(* IEC 61131-3 sources: AXOpen/src/components.elements/ctrl/test, 10 files *)

(* ---- AxoAiTests.st ---- *)
USING AxUnit;
USING AXOpen.Components.Elements;
USING AXOpen.Core;
USING AXOpen.Rtc;
USING AXOpen.Logging;

NAMESPACE AXOpen.Components.Elements.Tests

    {TestFixture}
    {S7.extern=ReadWrite}
    CLASS AxoAiTests
        VAR
            context : TestContext;
            _testAxoAi : AxoAi;
            _signal : DINT;

            _done : BOOL;
        END_VAR

        {Test(signal := 100, required := 100)}
        {Test(signal := 50, required := 50)}
        {Test(signal := 0, required := 0)}
        {Test(signal := -50, required := -50)}
        {Test(signal := -100, required := -100)}
        METHOD PUBLIC RoundedRawRoundedReal
            VAR_INPUT
                signal : DINT;
                required : REAL;
            END_VAR

            context.Open();

            _testAxoAi._config.RawLow := -100;
            _testAxoAi._config.RawHigh := 100;
            _testAxoAi._config.RealLow := -100;
            _testAxoAi._config.RealHigh := 100;
            _testAxoAi._config.Gain := 1;
            _testAxoAi._config.Offset := 0;
            _signal := signal;

            _testAxoAi.Run(context.SignalParent, _signal);

            AxUnit.Assert.Equal(TRUE, TO_DINT(required) = TO_DINT(_testAxoAi._scaled));

            context.Close();

        END_METHOD

        {Test(signal := 32767, required := 100)}
        {Test(signal := 16384, required := 50)}
        {Test(signal := 0, required := 0)}
        METHOD PUBLIC UnsignedRawTest
            VAR_INPUT
                signal : DINT;
                required : REAL;
            END_VAR

            context.Open();

            _testAxoAi._config.RawLow := 0;
            _testAxoAi._config.RawHigh := 32767;
            _testAxoAi._config.RealLow := 0;
            _testAxoAi._config.RealHigh := 100;
            _testAxoAi._config.Gain := 1;
            _testAxoAi._config.Offset := 0;
            _signal := signal;

            _testAxoAi.Run(context.SignalParent, _signal);

            AxUnit.Assert.Equal(TRUE, TO_DINT(required) = TO_DINT(_testAxoAi._scaled));

            context.Close();

        END_METHOD

        {Test(signal := 32767, required := 100)}
        {Test(signal := 0, required := 50)}
        {Test(signal := -32768, required := 0)}
        METHOD PUBLIC SignedRawTest
            VAR_INPUT
                signal : DINT;
                required : REAL;
            END_VAR

            context.Open();

            _testAxoAi._config.RawLow := -32768;
            _testAxoAi._config.RawHigh := 32767;
            _testAxoAi._config.RealLow := 0;
            _testAxoAi._config.RealHigh := 100;
            _testAxoAi._config.Gain := 1;
            _testAxoAi._config.Offset := 0;
            _signal := signal;

            _testAxoAi.Run(context.SignalParent, _signal);

            AxUnit.Assert.Equal(TRUE, TO_DINT(required) = TO_DINT(_testAxoAi._scaled));

            context.Close();

        END_METHOD

        {Test(signal := 32767, required := 100)}
        {Test(signal := 16384, required := 75)}
        {Test(signal := 0, required := 50)}
        METHOD PUBLIC UnsignedRaw_RealOffsetTest
            VAR_INPUT
                signal : DINT;
                required : REAL;
            END_VAR

            context.Open();

            _testAxoAi._config.RawLow := 0;
            _testAxoAi._config.RawHigh := 32767;
            _testAxoAi._config.RealLow := 50;
            _testAxoAi._config.RealHigh := 100;
            _testAxoAi._config.Gain := 1;
            _testAxoAi._config.Offset := 0;
            _signal := signal;

            _testAxoAi.Run(context.SignalParent, _signal);

            AxUnit.Assert.Equal(TRUE, TO_DINT(required) = TO_DINT(_testAxoAi._scaled));

            context.Close();

        END_METHOD

        {Test(signal := 32767, required := 100)}
        {Test(signal := 0, required := 75)}
        {Test(signal := -32768, required := 50)}
        METHOD PUBLIC SignedRaw_RealOffsetTest
            VAR_INPUT
                signal : DINT;
                required : REAL;
            END_VAR

            context.Open();

            _testAxoAi._config.RawLow := -32768;
            _testAxoAi._config.RawHigh := 32767;
            _testAxoAi._config.RealLow := 50;
            _testAxoAi._config.RealHigh := 100;
            _testAxoAi._config.Gain := 1;
            _testAxoAi._config.Offset := 0;
            _signal := signal;

            _testAxoAi.Run(context.SignalParent, _signal);

            AxUnit.Assert.Equal(TRUE, TO_DINT(required) = TO_DINT(_testAxoAi._scaled));

            context.Close();

        END_METHOD

        {Test(signal := 32767, required := 100)}
        {Test(signal := 16384, required := 0)}
        {Test(signal := 0, required := -100)}
        METHOD PUBLIC UnsignedRaw_RealSignedOffsetTest
            VAR_INPUT
                signal : DINT;
                required : REAL;
            END_VAR

            context.Open();

            _testAxoAi._config.RawLow := 0;
            _testAxoAi._config.RawHigh := 32767;
            _testAxoAi._config.RealLow := -100;
            _testAxoAi._config.RealHigh := 100;
            _testAxoAi._config.Gain := 1;
            _testAxoAi._config.Offset := 0;
            _signal := signal;

            _testAxoAi.Run(context.SignalParent, _signal);

            AxUnit.Assert.Equal(TRUE, TO_DINT(required) = TO_DINT(_testAxoAi._scaled));

            context.Close();

        END_METHOD

        {Test(signal := 32767, required := 100)}
        {Test(signal := 0, required := 0)}
        {Test(signal := -32768, required := -100)}
        METHOD PUBLIC SignedRaw_RealSignedOffsetTest
            VAR_INPUT
                signal : DINT;
                required : REAL;
            END_VAR

            context.Open();

            _testAxoAi._config.RawLow := -32768;
            _testAxoAi._config.RawHigh := 32767;
            _testAxoAi._config.RealLow := -100;
            _testAxoAi._config.RealHigh := 100;
            _testAxoAi._config.Gain := 1;
            _testAxoAi._config.Offset := 0;
            _signal := signal;

            _testAxoAi.Run(context.SignalParent, _signal);

            AxUnit.Assert.Equal(TRUE, TO_DINT(required) = TO_DINT(_testAxoAi._scaled));

            context.Close();

        END_METHOD

        {Test(signal := 32767, required := 120)}
        {Test(signal := 16384, required := 20)}
        {Test(signal := 0, required := -80)}
        METHOD PUBLIC UnSignedRaw_RealSignedOffset_WithOffsetCorrectionTest
            VAR_INPUT
                signal : DINT;
                required : REAL;
            END_VAR

            context.Open();

            _testAxoAi._config.RawLow := 0;
            _testAxoAi._config.RawHigh := 32767;
            _testAxoAi._config.RealLow := -100;
            _testAxoAi._config.RealHigh := 100;
            _testAxoAi._config.Gain := 1;
            _testAxoAi._config.Offset := 20;
            _signal := signal;

            _testAxoAi.Run(context.SignalParent, _signal);

            AxUnit.Assert.Equal(TRUE, TO_DINT(required) = TO_DINT(_testAxoAi._scaled));

            context.Close();

        END_METHOD

        {Test(signal := 32767, required := 120)}
        {Test(signal := 0, required := 20)}
        {Test(signal := -32768, required := -80)}
        METHOD PUBLIC SignedRaw_RealSignedOffset_WithOffsetCorrectionTest
            VAR_INPUT
                signal : DINT;
                required : REAL;
            END_VAR

            context.Open();

            _testAxoAi._config.RawLow := -32768;
            _testAxoAi._config.RawHigh := 32767;
            _testAxoAi._config.RealLow := -100;
            _testAxoAi._config.RealHigh := 100;
            _testAxoAi._config.Gain := 1;
            _testAxoAi._config.Offset := 20;
            _signal := signal;

            _testAxoAi.Run(context.SignalParent, _signal);

            AxUnit.Assert.Equal(TRUE, TO_DINT(required) = TO_DINT(_testAxoAi._scaled));

            context.Close();

        END_METHOD

    END_CLASS
END_NAMESPACE

(* ---- AxoAoTests.st ---- *)
USING AxUnit;
USING AXOpen.Components.Elements;
USING AXOpen.Core;
USING AXOpen.Rtc;
USING AXOpen.Logging;

NAMESPACE AXOpen.Components.Elements.Tests

    {TestFixture}
    {S7.extern=ReadWrite}
    CLASS AxoAoTests
        VAR
            context : TestContext;
            _testAxoAo : AxoAo;
            _signal : DINT;

            _unscaledResult : DINT;
        END_VAR

        {Test(required := 100, setVal := 100)}
        {Test(required := 50, setVal := 50)}
        {Test(required := 0, setVal := 0)}
        {Test(required := -50, setVal := -50)}
        {Test(required := -100, setVal := -100)}
        METHOD PUBLIC RoundedRawRoundedRealTest
            VAR_INPUT
                required : DINT;
                setVal : REAL;
            END_VAR

            context.Open();
            _signal := 0;

            _testAxoAo._config.RawLow := -100;
            _testAxoAo._config.RawHigh := 100;
            _testAxoAo._config.RealLow := -100;
            _testAxoAo._config.RealHigh := 100;
            _testAxoAo._config.Gain := 1;
            _testAxoAo._config.Offset := 0;

            _testAxoAo._requiredValue := setVal;

            _testAxoAo.Run(context.SignalParent, _signal);

            AxUnit.Assert.Equal(TRUE, required = TO_DINT(_testAxoAo._unscaled));
            AxUnit.Assert.Equal(TRUE, _signal = required);

            context.Close();

        END_METHOD

        {Test(required := 32767, setVal := 100, epsilon := 0)}
        {Test(required := REAL#16383.5, setVal := 50, epsilon := 1)}
        {Test(required := 0, setVal := 0, epsilon := 1)}

        METHOD PUBLIC UnsignedRawTest
            VAR_INPUT
                required : REAL;
                setVal : REAL;
                epsilon : DINT;
            END_VAR

            context.Open();
            _signal := 0;
            _unscaledResult := 0;
            _testAxoAo._config.RawLow := 0;
            _testAxoAo._config.RawHigh := 32767;
            _testAxoAo._config.RealLow := 0;
            _testAxoAo._config.RealHigh := 100;
            _testAxoAo._config.Gain := 1;
            _testAxoAo._config.Offset := 0;

            _testAxoAo._requiredValue := setVal;

            _testAxoAo.Run(context.SignalParent, _signal);
            _unscaledResult := TO_DINT(_testAxoAo._status.Unscaled);

            AxUnit.Assert.Equal(TRUE, TO_REAL(_unscaledResult - epsilon) <= required AND required <= TO_REAL(_unscaledResult + epsilon));
            AxUnit.Assert.Equal(TRUE, _signal = TO_DINT(required));

            context.Close();

        END_METHOD

        {Test(required := 32767, setVal := 100, epsilon := 0)}
        {Test(required := 0, setVal := 50, epsilon := 1)}
        {Test(required := -32768, setVal := 0, epsilon := 1)}

        METHOD PUBLIC SignedRawTest
            VAR_INPUT
                required : REAL;
                setVal : REAL;
                epsilon : DINT;
            END_VAR

            context.Open();
            _signal := 0;
            _testAxoAo._status.Unscaled := 0;
            _testAxoAo._config.RawLow := -32768;
            _testAxoAo._config.RawHigh := 32767;
            _testAxoAo._config.RealLow := 0;
            _testAxoAo._config.RealHigh := 100;
            _testAxoAo._config.Gain := 1;
            _testAxoAo._config.Offset := 0;

            _testAxoAo._requiredValue := setVal;

            _testAxoAo.Run(context.SignalParent, _signal);
            _unscaledResult := TO_DINT(_testAxoAo._status.Unscaled);
            AxUnit.Assert.Equal(TRUE, TO_REAL(_unscaledResult - epsilon) <= required AND required <= TO_REAL(_unscaledResult + epsilon));
            AxUnit.Assert.Equal(TRUE, _signal = TO_DINT(required));

            context.Close();

        END_METHOD

        {Test(required := 32767, setVal := 100, epsilon := 0)}
        {Test(required := REAL#16383.5, setVal := 75, epsilon := 1)}
        {Test(required := 0, setVal := 50, epsilon := 0)}
        METHOD PUBLIC UnSignedRawTest_RealOffsetTest
            VAR_INPUT
                required : REAL;
                setVal : REAL;
                epsilon : DINT;
            END_VAR

            context.Open();
            _signal := 0;
            _unscaledResult := 0;
            _testAxoAo._config.RawLow := 0;
            _testAxoAo._config.RawHigh := 32767;
            _testAxoAo._config.RealLow := 50;
            _testAxoAo._config.RealHigh := 100;
            _testAxoAo._config.Gain := 1;
            _testAxoAo._config.Offset := 0;

            _testAxoAo._requiredValue := setVal;

            _testAxoAo.Run(context.SignalParent, _signal);
            _unscaledResult := TO_DINT(_testAxoAo._status.Unscaled);
            AxUnit.Assert.Equal(TRUE, TO_REAL(_unscaledResult - epsilon) <= required AND required <= TO_REAL(_unscaledResult + epsilon));
            AxUnit.Assert.Equal(TRUE, _signal = TO_DINT(required));

            context.Close();

        END_METHOD

        {Test(required := 32767, setVal := 100, epsilon := 0)}
        {Test(required := 0, setVal := 75, epsilon := 1)}
        {Test(required := -32768, setVal := 50, epsilon := 0)}
        METHOD PUBLIC SignedRawTest_RealOffsetTest
            VAR_INPUT
                required : REAL;
                setVal : REAL;
                epsilon : DINT;
            END_VAR

            context.Open();
            _signal := 0;
            _unscaledResult := 0;
            _testAxoAo._config.RawLow := -32768;
            _testAxoAo._config.RawHigh := 32767;
            _testAxoAo._config.RealLow := 50;
            _testAxoAo._config.RealHigh := 100;
            _testAxoAo._config.Gain := 1;
            _testAxoAo._config.Offset := 0;

            _testAxoAo._requiredValue := setVal;

            _testAxoAo.Run(context.SignalParent, _signal);
            _unscaledResult := TO_DINT(_testAxoAo._status.Unscaled);
            AxUnit.Assert.Equal(TRUE, TO_REAL(_unscaledResult - epsilon) <= required AND required <= TO_REAL(_unscaledResult + epsilon));
            AxUnit.Assert.Equal(TRUE, _signal = TO_DINT(required));

            context.Close();

        END_METHOD

        {Test(required := 32767, setVal := 100, epsilon := 0)}
        {Test(required := 16384, setVal := 0, epsilon := 2)}
        {Test(required := 0, setVal := -100, epsilon := 0)}
        METHOD PUBLIC UnsignedRawTest_RealSignedOffsetTest
            VAR_INPUT
                required : REAL;
                setVal : REAL;
                epsilon : DINT;
            END_VAR

            context.Open();
            _signal := 0;
            _unscaledResult := 0;
            _testAxoAo._config.RawLow := 0;
            _testAxoAo._config.RawHigh := 32767;
            _testAxoAo._config.RealLow := -100;
            _testAxoAo._config.RealHigh := 100;
            _testAxoAo._config.Gain := 1;
            _testAxoAo._config.Offset := 0;

            _testAxoAo._requiredValue := setVal;

            _testAxoAo.Run(context.SignalParent, _signal);
            _unscaledResult := TO_DINT(_testAxoAo._status.Unscaled);
            AxUnit.Assert.Equal(TRUE, TO_REAL(_unscaledResult - epsilon) <= required AND required <= TO_REAL(_unscaledResult + epsilon));
            AxUnit.Assert.Equal(TRUE, _signal = TO_DINT(required));

            context.Close();

        END_METHOD

        {Test(required := 32767, setVal := 100, epsilon := 0)}
        {Test(required := 0, setVal := 0, epsilon := 1)}
        {Test(required := -32768, setVal := -100, epsilon := 0)}
        METHOD PUBLIC SignedRawTest_RealSignedOffsetTest
            VAR_INPUT
                required : REAL;
                setVal : REAL;
                epsilon : DINT;
            END_VAR

            context.Open();
            _signal := 0;
            _unscaledResult := 0;
            _testAxoAo._config.RawLow := -32768;
            _testAxoAo._config.RawHigh := 32767;
            _testAxoAo._config.RealLow := -100;
            _testAxoAo._config.RealHigh := 100;
            _testAxoAo._config.Gain := 1;
            _testAxoAo._config.Offset := 0;

            _testAxoAo._requiredValue := setVal;

            _testAxoAo.Run(context.SignalParent, _signal);
            _unscaledResult := TO_DINT(_testAxoAo._status.Unscaled);
            AxUnit.Assert.Equal(TRUE, TO_REAL(_unscaledResult - epsilon) <= required AND required <= TO_REAL(_unscaledResult + epsilon));
            AxUnit.Assert.Equal(TRUE, _signal = TO_DINT(required));

            context.Close();

        END_METHOD

        {Test(required := REAL#32787.0, setVal := 100, epsilon := 0)}
        {Test(required := 16404, setVal := 0, epsilon := 1)}
        {Test(required := 20, setVal := -100, epsilon := 0)}
        METHOD PUBLIC UnSignedRawTest_RealSignedOffset_WithOffsetCorrectionTest
            VAR_INPUT

                required : REAL;
                setVal : REAL;
                epsilon : DINT;
            END_VAR

            context.Open();
            _signal := 0;
            _unscaledResult := 0;
            _testAxoAo._config.RawLow := 0;
            _testAxoAo._config.RawHigh := 32767;
            _testAxoAo._config.RealLow := -100;
            _testAxoAo._config.RealHigh := 100;
            _testAxoAo._config.Gain := 1;
            _testAxoAo._config.Offset := 20;

            _testAxoAo._requiredValue := setVal;

            _testAxoAo.Run(context.SignalParent, _signal);

            _unscaledResult := TO_DINT(_testAxoAo._status.Unscaled);
            AxUnit.Assert.Equal(TRUE, TO_REAL(_unscaledResult - epsilon) <= required AND required <= TO_REAL(_unscaledResult + epsilon));
            AxUnit.Assert.Equal(TRUE, _signal = TO_DINT(required));

            context.Close();

        END_METHOD

        {Test(required := REAL#32787.0, setVal := 100, epsilon := 0)}
        {Test(required := 16404, setVal := 0, epsilon := 1)}
        {Test(required := 20, setVal := -100, epsilon := 0)}
        METHOD PUBLIC SignedRawTest_RealSignedOffset_WithOffsetCorrectionTest
            VAR_INPUT
                required : REAL;
                setVal : REAL;
                epsilon : DINT;
            END_VAR

            context.Open();
            _signal := 0;
            _unscaledResult := 0;
            _testAxoAo._config.RawLow := 0;
            _testAxoAo._config.RawHigh := 32767;
            _testAxoAo._config.RealLow := -100;
            _testAxoAo._config.RealHigh := 100;
            _testAxoAo._config.Gain := 1;
            _testAxoAo._config.Offset := 20;

            _testAxoAo._requiredValue := setVal;

            _testAxoAo.Run(context.SignalParent, _signal);

            _unscaledResult := TO_DINT(_testAxoAo._status.Unscaled);
            AxUnit.Assert.Equal(TRUE, TO_REAL(_unscaledResult - epsilon) <= required AND required <= TO_REAL(_unscaledResult + epsilon));
            AxUnit.Assert.Equal(TRUE, _signal = TO_DINT(required));

            context.Close();

        END_METHOD

    END_CLASS
END_NAMESPACE

(* ---- AxoButtonWithIndicatorTests.st ---- *)
USING AxUnit;
USING AXOpen.Components.Elements;
USING AXOpen.Core;
USING AXOpen.Rtc;
USING AXOpen.Logging;
USING AXOpen.Components.Elements;

NAMESPACE AXOpen.Components.Elements.Tests

    {TestFixture}
    {S7.extern=ReadWrite}
    CLASS AxoButtonWithIndicatorTests
        VAR
            context : TestContext;
            _testButtonWithIndicator : AxoBacklitButton;
            _inputSignal : BOOL;
            _ledOutput : BOOL;
        END_VAR

        {Test}
        METHOD PUBLIC Test_Run_all_on
            VAR
                signal : BOOL := TRUE;
            END_VAR

            context.Open();
            _inputSignal := TRUE;
            _testButtonWithIndicator.Run(context.SignalParent, _inputSignal, _ledOutput);

            // Assert that the button component processes the signal correctly
            AxUnit.Assert.Equal(TRUE, _testButtonWithIndicator.Button.IsTrue());
            _testButtonWithIndicator.Led.Set();
            AxUnit.Assert.Equal(TRUE, _testButtonWithIndicator.Led.IsTrue());
            context.Close();
        END_METHOD

        {Test}
        METHOD PUBLIC Test_Run_all_off
            VAR
                signal : BOOL := TRUE;
            END_VAR

            context.Open();
            _inputSignal := FALSE;
            _testButtonWithIndicator.Run(context.SignalParent, _inputSignal, _ledOutput);

            // Assert that the button component processes the signal correctly
            AxUnit.Assert.Equal(TRUE, _testButtonWithIndicator.Button.IsFalse());
            _testButtonWithIndicator.Led.Reset();
            AxUnit.Assert.Equal(TRUE, _testButtonWithIndicator.Led.IsFalse());
            context.Close();
        END_METHOD

        {Test}
        METHOD PUBLIC Test_Run_NullParent_DoesNotRun
            VAR
                signal : BOOL := TRUE;
            END_VAR

            _inputSignal := TRUE;
            _testButtonWithIndicator.Run(NULL, _inputSignal, _ledOutput);

            // Assert that nothing happens when inParent is null
            // The component should not process anything

        END_METHOD

        {Test}
        METHOD PUBLIC Test_Restore_CallsRestoreOnChildren
            context.Open();
            _testButtonWithIndicator.Restore();
            context.Close();
        END_METHOD

        {Test}
        METHOD PUBLIC Test_ManualControl_CallsManualControlOnChildren
            context.Open();
            _testButtonWithIndicator.ActivateManualControl();
            context.Close();
        END_METHOD
    END_CLASS
END_NAMESPACE

(* ---- AxoDiTests.st ---- *)
USING AxUnit;
USING AXOpen.Elements;
USING AXOpen.Core;
USING AXOpen.Rtc;
USING AXOpen.Logging;

NAMESPACE AXOpen.Elements.Tests

    {TestFixture}
    {S7.extern=ReadWrite}
    CLASS AxoDiTests
        VAR
            context : TestContext;
            _testAxoDi : AxoDi;
            _signal : BOOL;

            _done : BOOL;
        END_VAR

        {Test}
        METHOD PUBLIC CheckForSignalStatusTrue

            context.Open();
            _signal := TRUE;
            _testAxoDi.Run(context.SignalParent, _signal);

            AxUnit.Assert.Equal(TRUE, _testAxoDi.IsTrue());
            AxUnit.Assert.Equal(FALSE, _testAxoDi.IsFalse());

            context.Close();

        END_METHOD

        {Test}
        METHOD PUBLIC CheckForSignalStatusFalse

            context.Open();
            _signal := FALSE;
            _testAxoDi.Run(context.SignalParent,_signal);

            AxUnit.Assert.Equal(FALSE, _testAxoDi.IsTrue());
            AxUnit.Assert.Equal(TRUE, _testAxoDi.IsFalse());

            context.Close();

        END_METHOD

    END_CLASS
END_NAMESPACE

(* ---- AxoDoTests.st ---- *)
USING AxUnit;
USING AXOpen.Components.Elements;
USING AXOpen.Core;
USING AXOpen.Rtc;
USING AXOpen.Logging;

NAMESPACE AXOpen.Components.Elements.Tests

    {TestFixture}
    {S7.extern=ReadWrite}
    CLASS AxoDoTests
        VAR
            context : TestContext;
            _testAxoDo : AxoDo;
            _signal : BOOL;

            _done : BOOL;
        END_VAR

        {Test}
        METHOD PUBLIC SetSignalOn

            context.Open();
            _testAxoDo.Run(context.SignalParent,_signal);
            _testAxoDo.Set();

            AxUnit.Assert.Equal(TRUE, _testAxoDo.IsTrue());
            AxUnit.Assert.Equal(FALSE, _testAxoDo.IsFalse());

            context.Close();

        END_METHOD

        {Test}
        METHOD PUBLIC SetSignalOff

            context.Open();
            _signal := TRUE;
            _testAxoDo.Run(context.SignalParent,_signal);
            _testAxoDo.Reset();

            AxUnit.Assert.Equal(FALSE, _testAxoDo.IsTrue());
            AxUnit.Assert.Equal(TRUE, _testAxoDo.IsFalse());

            context.Close();

        END_METHOD

    END_CLASS
END_NAMESPACE

(* ---- AxoLightColumnTests.st ---- *)
USING AxUnit;
USING AXOpen.Elements;
USING AXOpen.Core;
USING AXOpen.Rtc;
USING AXOpen.Logging;
USING AXOpen.Components.Elements;

NAMESPACE AXOpen.Elements.Tests

    {TestFixture}
    {S7.extern=ReadWrite}
    CLASS AxoLightColumnTests
        VAR
            context : TestContext;
            _testLightColumn : AxoLightColumn;
            _redOutput : BOOL;
            _greenOutput : BOOL;
            _blueOutput : BOOL;
            _yellowOutput : BOOL;
            _hornOutput : BOOL;
        END_VAR

        {Test}
        METHOD PUBLIC Test_Run_WithValidParent
            context.Open();

            _testLightColumn.Run(inParent := context.SignalParent, oRed => _redOutput, oGreen => _greenOutput, oBlue => _blueOutput, oYellow => _yellowOutput, oHorn => _hornOutput);

            // Test that the component runs without errors when parent is valid
            // The outputs should be processed correctly
            context.Close();
        END_METHOD

        {Test}
        METHOD PUBLIC Test_Run_NullParent_DoesNotRun
            _testLightColumn.Run(inParent := NULL, oRed => _redOutput, oGreen => _greenOutput, oBlue => _blueOutput, oYellow => _yellowOutput, oHorn => _hornOutput);

            // Component should not process anything when parent is null
            // No exceptions should be thrown
        END_METHOD

        {Test}
        METHOD PUBLIC Test_Red_SetAndReset
            context.Open();

            // Set red light
            _testLightColumn.Red.Set();
            _testLightColumn.Run(inParent := context.SignalParent, oRed => _redOutput, oGreen => _greenOutput, oBlue => _blueOutput, oYellow => _yellowOutput, oHorn => _hornOutput);

            AxUnit.Assert.Equal(TRUE, _testLightColumn.Red.IsTrue());

            // Reset red light
            _testLightColumn.Red.Reset();
            _testLightColumn.Run(inParent := context.SignalParent, oRed => _redOutput, oGreen => _greenOutput, oBlue => _blueOutput, oYellow => _yellowOutput, oHorn => _hornOutput);

            AxUnit.Assert.Equal(FALSE, _testLightColumn.Red.IsTrue());

            context.Close();
        END_METHOD

        {Test}
        METHOD PUBLIC Test_Green_SetAndReset
            context.Open();

            // Set green light
            _testLightColumn.Green.Set();
            _testLightColumn.Run(inParent := context.SignalParent, oRed => _redOutput, oGreen => _greenOutput, oBlue => _blueOutput, oYellow => _yellowOutput, oHorn => _hornOutput);

            AxUnit.Assert.Equal(TRUE, _testLightColumn.Green.IsTrue());

            // Reset green light
            _testLightColumn.Green.Reset();
            _testLightColumn.Run(inParent := context.SignalParent, oRed => _redOutput, oGreen => _greenOutput, oBlue => _blueOutput, oYellow => _yellowOutput, oHorn => _hornOutput);

            AxUnit.Assert.Equal(FALSE, _testLightColumn.Green.IsTrue());

            context.Close();
        END_METHOD

        {Test}
        METHOD PUBLIC Test_Blue_SetAndReset
            context.Open();

            // Set blue light
            _testLightColumn.Blue.Set();
            _testLightColumn.Run(inParent := context.SignalParent, oRed => _redOutput, oGreen => _greenOutput, oBlue => _blueOutput, oYellow => _yellowOutput, oHorn => _hornOutput);

            AxUnit.Assert.Equal(TRUE, _testLightColumn.Blue.IsTrue());

            // Reset blue light
            _testLightColumn.Blue.Reset();
            _testLightColumn.Run(inParent := context.SignalParent, oRed => _redOutput, oGreen => _greenOutput, oBlue => _blueOutput, oYellow => _yellowOutput, oHorn => _hornOutput);

            AxUnit.Assert.Equal(FALSE, _testLightColumn.Blue.IsTrue());

            context.Close();
        END_METHOD

        {Test}
        METHOD PUBLIC Test_Yellow_SetAndReset
            context.Open();

            // Set yellow light
            _testLightColumn.Yellow.Set();
            _testLightColumn.Run(inParent := context.SignalParent, oRed => _redOutput, oGreen => _greenOutput, oBlue => _blueOutput, oYellow => _yellowOutput, oHorn => _hornOutput);

            AxUnit.Assert.Equal(TRUE, _testLightColumn.Yellow.IsTrue());

            // Reset yellow light
            _testLightColumn.Yellow.Reset();
            _testLightColumn.Run(inParent := context.SignalParent, oRed => _redOutput, oGreen => _greenOutput, oBlue => _blueOutput, oYellow => _yellowOutput, oHorn => _hornOutput);

            AxUnit.Assert.Equal(FALSE, _testLightColumn.Yellow.IsTrue());

            context.Close();
        END_METHOD

        {Test}
        METHOD PUBLIC Test_Horn_SetAndReset
            context.Open();

            // Set horn
            _testLightColumn.Horn.Set();
            _testLightColumn.Run(inParent := context.SignalParent, oRed => _redOutput, oGreen => _greenOutput, oBlue => _blueOutput, oYellow => _yellowOutput, oHorn => _hornOutput);

            AxUnit.Assert.Equal(TRUE, _testLightColumn.Horn.IsTrue());

            // Reset horn
            _testLightColumn.Horn.Reset();
            _testLightColumn.Run(inParent := context.SignalParent, oRed => _redOutput, oGreen => _greenOutput, oBlue => _blueOutput, oYellow => _yellowOutput, oHorn => _hornOutput);

            AxUnit.Assert.Equal(FALSE, _testLightColumn.Horn.IsTrue());

            context.Close();
        END_METHOD

        {Test}
        METHOD PUBLIC Test_MultipleLights_SetSimultaneously
            context.Open();

            // Set multiple lights at once
            _testLightColumn.Red.Set();
            _testLightColumn.Green.Set();
            _testLightColumn.Horn.Set();

            _testLightColumn.Run(inParent := context.SignalParent, oRed => _redOutput, oGreen => _greenOutput, oBlue => _blueOutput, oYellow => _yellowOutput, oHorn => _hornOutput);

            AxUnit.Assert.Equal(TRUE, _testLightColumn.Red.IsTrue());
            AxUnit.Assert.Equal(TRUE, _testLightColumn.Green.IsTrue());
            AxUnit.Assert.Equal(FALSE, _testLightColumn.Blue.IsTrue());
            AxUnit.Assert.Equal(FALSE, _testLightColumn.Yellow.IsTrue());
            AxUnit.Assert.Equal(TRUE, _testLightColumn.Horn.IsTrue());

            context.Close();
        END_METHOD

        {Test}
        METHOD PUBLIC Test_Restore_CallsRestoreOnAllComponents
            context.Open();

            // Set some lights first
            _testLightColumn.Red.Set();
            _testLightColumn.Green.Reset();
            _testLightColumn.Blue.Reset();
            _testLightColumn.Yellow.Set();
            _testLightColumn.Horn.Set();

            // Now restore
            _testLightColumn.Restore();

            // After restore, the signals should maintain the previous state since only tasks are restored.
            _testLightColumn.Run(inParent := context.SignalParent, oRed => _redOutput, oGreen => _greenOutput, oBlue => _blueOutput, oYellow => _yellowOutput, oHorn => _hornOutput);

            AxUnit.Assert.Equal(TRUE, _testLightColumn.Red.IsTrue());
            AxUnit.Assert.Equal(TRUE, _testLightColumn.Green.IsFalse());
            AxUnit.Assert.Equal(TRUE, _testLightColumn.Blue.IsFalse());
            AxUnit.Assert.Equal(TRUE, _testLightColumn.Yellow.IsTrue());
            AxUnit.Assert.Equal(TRUE, _testLightColumn.Horn.IsTrue());

            context.Close();
        END_METHOD

        {Test}
        METHOD PUBLIC Test_AllLights_Off_Initially
            context.Open();

            // Test that all lights start in OFF state
            _testLightColumn.Run(inParent := context.SignalParent, oRed => _redOutput, oGreen => _greenOutput, oBlue => _blueOutput, oYellow => _yellowOutput, oHorn => _hornOutput);

            AxUnit.Assert.Equal(FALSE, _testLightColumn.Red.IsTrue());
            AxUnit.Assert.Equal(FALSE, _testLightColumn.Green.IsTrue());
            AxUnit.Assert.Equal(FALSE, _testLightColumn.Blue.IsTrue());
            AxUnit.Assert.Equal(FALSE, _testLightColumn.Yellow.IsTrue());
            AxUnit.Assert.Equal(FALSE, _testLightColumn.Horn.IsTrue());

            context.Close();
        END_METHOD
    END_CLASS
END_NAMESPACE

(* ---- AxoLockDoorWithSensorTests.st ---- *)
USING AxUnit;
USING AXOpen.Elements;
USING AXOpen.Core;
USING AXOpen.Rtc;
USING AXOpen.Logging;
USING AXOpen.Components.Elements;

NAMESPACE AXOpen.Elements.Tests

    {TestFixture}
    {S7.extern=ReadWrite}
    CLASS AxoLockDoorWithSensorTests
        VAR
            context : TestContext;
            _testDoorLock : AxoDoorLockWithSensor;
            _isLockOpen : BOOL;
            _isSensorOpen : BOOL;
            _isLocked : BOOL;
            _lockOutput : BOOL;
            _lockResult : BOOL;
            _unlockResult : BOOL;
            _isClosedResult : BOOL;
        END_VAR

        {Test}
        METHOD PUBLIC Test_Run_WithValidParent
            context.Open();
            _isLockOpen := FALSE;
            _isSensorOpen := FALSE;
            _isLocked := TRUE;

            _testDoorLock.Run(context.SignalParent, _isLockOpen, _isSensorOpen, _isLocked, _lockOutput);

            // Assert that inputs are processed correctly
            AxUnit.Assert.Equal(FALSE, _testDoorLock.IsLockOpen.IsTrue());
            AxUnit.Assert.Equal(FALSE, _testDoorLock.IsSensorOpen.IsTrue());
            AxUnit.Assert.Equal(TRUE, _testDoorLock._IsLocked);

            context.Close();
        END_METHOD

        {Test}
        METHOD PUBLIC Test_Run_NullParent_DoesNotRun
            _isLockOpen := FALSE;
            _isSensorOpen := FALSE;
            _isLocked := TRUE;

            _testDoorLock.Run(NULL, _isLockOpen, _isSensorOpen, _isLocked, _lockOutput);

            // Component should not process anything when parent is null
        END_METHOD

        {Test}
        METHOD PUBLIC Test_Lock_DoorClosedAndLocked_ReturnsTrue
            context.Open();
            _isLockOpen := FALSE;
            _isSensorOpen := FALSE;
            _isLocked := TRUE;

            _testDoorLock.Run(context.SignalParent, _isLockOpen, _isSensorOpen, _isLocked, _lockOutput);

            _lockResult := _testDoorLock.Lock();

            AxUnit.Assert.Equal(TRUE, _lockResult);

            context.Close();
        END_METHOD

        {Test}
        METHOD PUBLIC Test_Lock_DoorOpenOrUnlocked_ReturnsFalse
            context.Open();
            _isLockOpen := TRUE; // Door is open
            _isSensorOpen := FALSE;
            _isLocked := FALSE; // Not locked

            _testDoorLock.Run(context.SignalParent, _isLockOpen, _isSensorOpen, _isLocked, _lockOutput);

            _lockResult := _testDoorLock.Lock();

            AxUnit.Assert.Equal(FALSE, _lockResult);

            context.Close();
        END_METHOD

        {Test}
        METHOD PUBLIC Test_UnLock_LockedDoor_ReturnsTrue
            context.Open();
            _isLockOpen := FALSE;
            _isSensorOpen := FALSE;
            _isLocked := FALSE; // Not locked

            _testDoorLock.Run(context.SignalParent, _isLockOpen, _isSensorOpen, _isLocked, _lockOutput);

            _unlockResult := _testDoorLock.UnLock();

            AxUnit.Assert.Equal(TRUE, _unlockResult);

            context.Close();
        END_METHOD

        {Test}
        METHOD PUBLIC Test_UnLock_AlreadyLocked_ReturnsFalse
            context.Open();
            _isLockOpen := FALSE;
            _isSensorOpen := FALSE;
            _isLocked := TRUE; // Already locked

            _testDoorLock.Run(context.SignalParent, _isLockOpen, _isSensorOpen, _isLocked, _lockOutput);

            _unlockResult := _testDoorLock.UnLock();

            AxUnit.Assert.Equal(FALSE, _unlockResult);

            context.Close();
        END_METHOD

        {Test}
        METHOD PUBLIC Test_IsClosed_BothSensorsClosed_ReturnsTrue
            context.Open();
            _isLockOpen := FALSE;
            _isSensorOpen := FALSE;
            _isLocked := TRUE;

            _testDoorLock.Run(context.SignalParent, _isLockOpen, _isSensorOpen, _isLocked, _lockOutput);

            _isClosedResult := _testDoorLock.IsClosed();

            AxUnit.Assert.Equal(TRUE, _isClosedResult);

            context.Close();
        END_METHOD

        {Test}
        METHOD PUBLIC Test_IsClosed_AnySensorOpen_ReturnsFalse
            context.Open();
            _isLockOpen := TRUE; // Lock sensor is open
            _isSensorOpen := FALSE;
            _isLocked := TRUE;

            _testDoorLock.Run(context.SignalParent, _isLockOpen, _isSensorOpen, _isLocked, _lockOutput);

            _isClosedResult := _testDoorLock.IsClosed();

            AxUnit.Assert.Equal(FALSE, _isClosedResult);

            context.Close();
        END_METHOD

        {Test}
        METHOD PUBLIC Test_Restore_CallsRestoreOnChildren
            context.Open();
            _testDoorLock.Restore();
            context.Close();
        END_METHOD
    END_CLASS
END_NAMESPACE

(* ---- AxoRotaryIndexingTableTests.st ---- *)
USING AxUnit;
USING AXOpen.Components.Elements;
USING AXOpen.Core;
USING AXOpen.Rtc;
USING AXOpen.Logging;

NAMESPACE AXOpen.Components.Elements.Tests

    {TestFixture}
    {S7.extern=ReadWrite}
    CLASS AxoRotaryIndexingTableTests
        VAR
            context : TestContext;
            _uut : AxoRotaryIndexingTable;
            _enableTurn : BOOL;
            _startTurn : BOOL;
            _configDefaults : AxoRotaryIndexingTable_Config;
            _stateDefaults : AxoRotaryIndexingTable_State;
            _controlDefaults : AxoRotaryIndexingTable_Control;
            _statusDefaults : AxoRotaryIndexingTable_Component_Status;
        END_VAR

        {Test}
        METHOD PUBLIC Config_DefaultValues

            AxUnit.Assert.Equal(LT#5S, _configDefaults.InfoTime);
            AxUnit.Assert.Equal(LT#10S, _configDefaults.ErrorTime);
            AxUnit.Assert.Equal(LT#10S, _configDefaults.TaskTimeout);
            AxUnit.Assert.Equal(TRUE, _configDefaults.Direction = eAxoRotaryIndexingTableDirection#Cw);
            AxUnit.Assert.Equal(UINT#0, _configDefaults.NumberOfPositions);
            AxUnit.Assert.Equal(UINT#0, _configDefaults.Offset);
        END_METHOD

        {Test}
        METHOD PUBLIC State_DefaultValues

            AxUnit.Assert.Equal(FALSE, _stateDefaults.SafetyCondition);
            AxUnit.Assert.Equal(FALSE, _stateDefaults.InPosition);
            AxUnit.Assert.Equal(FALSE, _stateDefaults.InPrecisePosition);
            AxUnit.Assert.Equal(UINT#0, _stateDefaults.CodingPosition);
        END_METHOD

        {Test}
        METHOD PUBLIC Control_DefaultValues

            AxUnit.Assert.Equal(FALSE, _controlDefaults.EnableTurn);
            AxUnit.Assert.Equal(FALSE, _controlDefaults.StartTurn);
        END_METHOD

        {Test}
        METHOD PUBLIC ComponentStatus_DefaultValues

            AxUnit.Assert.Equal(UINT#0, _statusDefaults.StartPosition);
            AxUnit.Assert.Equal(UINT#0, _statusDefaults.EndPosition);
            AxUnit.Assert.Equal(UINT#0, _statusDefaults.Positions[0]);
            AxUnit.Assert.Equal(UINT#0, _statusDefaults.Positions[16]);
            AxUnit.Assert.Equal(UINT#0, _statusDefaults.Positions[32]);
        END_METHOD

        {Test}
        METHOD PUBLIC Run_WithNullParent_SetsProgrammingError
            _uut.Config.NumberOfPositions := UINT#4;
            _uut.Run(NULL, TRUE, TRUE, TRUE, UINT#1, _enableTurn, _startTurn);

            AxUnit.Assert.Equal(UINT#700, _uut.Status.Error.Id);
        END_METHOD

        {Test}
        METHOD PUBLIC Run_WithTooFewPositions_SetsProgrammingError
            context.Open();
            _enableTurn := FALSE;
            _startTurn := FALSE;
            _uut.Config.NumberOfPositions := UINT#1;

            _uut.Run(context.SignalParent, TRUE, TRUE, TRUE, UINT#1, _enableTurn, _startTurn);

            AxUnit.Assert.Equal(UINT#701, _uut.Status.Error.Id);
            context.Close();
        END_METHOD

        METHOD PUBLIC Run_WithZeroOffset_DefaultsToOne
            context.Open();
            _enableTurn := FALSE;
            _startTurn := FALSE;
            _uut.Config.NumberOfPositions := UINT#4;
            _uut.Config.Offset := UINT#0;

            _uut.Run(context.SignalParent, TRUE, TRUE, TRUE, UINT#2, _enableTurn, _startTurn);

            AxUnit.Assert.Equal(UINT#1, _uut.Config.Offset);
            AxUnit.Assert.Equal(UINT#0, _uut.Status.Error.Id);
            context.Close();
        END_METHOD

        {Test}
        METHOD PUBLIC Run_ComputesPositionsAndCurrentPosition
            context.Open();
            _enableTurn := FALSE;
            _startTurn := FALSE;
            _uut.Config.NumberOfPositions := UINT#4;
            _uut.Config.Offset := UINT#1;

            _uut.Run(context.SignalParent, TRUE, TRUE, TRUE, UINT#3, _enableTurn, _startTurn);

            AxUnit.Assert.Equal(UINT#3, _uut.CurrentPosition);
            AxUnit.Assert.Equal(UINT#0, _uut.Status.Error.Id);
            AxUnit.Assert.Equal(UINT#3, _uut.Status.Positions[0]);
            AxUnit.Assert.Equal(UINT#2, _uut.Status.Positions[1]);
            AxUnit.Assert.Equal(UINT#1, _uut.Status.Positions[2]);
            AxUnit.Assert.Equal(UINT#4, _uut.Status.Positions[3]);
            AxUnit.Assert.Equal(FALSE, _enableTurn);
            AxUnit.Assert.Equal(FALSE, _startTurn);
            context.Close();
        END_METHOD

        {Test}
        METHOD PUBLIC Restore_ResetsOutputsAndStatus
            _uut.Status.Error.Id := UINT#999;
            _uut.Status.Action.Id := UINT#555;
            _uut.Outputs.EnableTurn := TRUE;
            _uut.Outputs.StartTurn := TRUE;

            _uut.Restore();

            AxUnit.Assert.Equal(UINT#0, _uut.Status.Error.Id);
            AxUnit.Assert.Equal(UINT#50, _uut.Status.Action.Id);
            AxUnit.Assert.Equal(FALSE, _uut.Outputs.EnableTurn);
            AxUnit.Assert.Equal(FALSE, _uut.Outputs.StartTurn);
        END_METHOD

    END_CLASS
END_NAMESPACE

(* ---- Mock.st ---- *)
USING AXOpen.Core;
USING AXOpen.Rtc;
USING AXOpen.Logging;
NAMESPACE AxoIO.Tests
    {S7.extern=ReadWrite}
    CLASS INTERNAL AxoRtcMock IMPLEMENTS IAxoRtc
        VAR PRIVATE
            _NowUTC : LDATE_AND_TIME;
        END_VAR

        METHOD INTERNAL SetNowUTC : LDATE_AND_TIME
            VAR_INPUT
                Set :  LDATE_AND_TIME;
            END_VAR;
            _NowUTC := Set;
        END_METHOD

        METHOD PUBLIC NowUTC : LDATE_AND_TIME
            NowUTC := _NowUTC;
        END_METHOD
    END_CLASS

    {S7.extern=ReadWrite}
    CLASS INTERNAL AxoLoggerMock IMPLEMENTS AXOpen.Logging.IAxoLogger
        VAR PUBLIC

        END_VAR

        /// <summary>
        /// Log method that captures a message, logging level, and the sender of the log.
        /// </summary>
        /// <param name="_message">The message to be logged.</param>
        /// <param name="_level">The severity level of the log.</param>
        /// <param name="_sender">The object that sends the log.</param>
        METHOD PUBLIC Log
            VAR_INPUT
                _message : STRING[254];
                _level : eLogLevel;
                _sender : IAxoObject;
            END_VAR

          ;
        END_METHOD

        /// <summary>
        /// Log method that captures a message and logging level.
        /// </summary>
        /// <param name="_message">The message to be logged.</param>
        /// <param name="_level">The severity level of the log.</param>
        METHOD PUBLIC Log
            VAR_INPUT
                _message : STRING[254];
                _level : eLogLevel;
            END_VAR

           ;
        END_METHOD

        /// <summary>
        /// Sets the minimum logging level to be captured by this logger.
        /// </summary>
        /// <param name="_level">The minimum log level.</param>
        /// <returns>Returns the instance of the logger.</returns>
        METHOD PUBLIC SetMinimumLevel : IAxoLoggerConfig
            VAR_INPUT
                _level : eLogLevel;
            END_VAR
            ;
        END_METHOD
    END_CLASS
END_NAMESPACE

(* ---- TestContext.st ---- *)
USING AXOpen.Core;
USING AXOpen.Rtc;
USING AXOpen.Logging;

NAMESPACE AxoIO.Tests
    {S7.extern=ReadWrite}
    CLASS TestContext EXTENDS AXOpen.Core.Dummies.MockAxoContext

        VAR PUBLIC
            SignalParent : AxoObject;
        END_VAR

        METHOD PUBLIC OVERRIDE Open : ULINT
            SUPER.Open();
            THIS.InitializeRootObject(SignalParent);
        END_METHOD

        METHOD PROTECTED OVERRIDE Main
               ;
        END_METHOD
    END_CLASS
END_NAMESPACE
